FUNCTION_BLOCK FB_LogicSupply
VAR_IN_OUT
	bSwitchOn		: BOOL;
END_VAR

{attribute 'TcRpcEnable'}
METHOD SwitchOff
bSwitchOn := FALSE;
END_METHOD

{attribute 'TcRpcEnable'}
METHOD SwitchOn
bSwitchOn := TRUE;
END_METHOD

END_FUNCTION_BLOCK

(* stored: Version 1.1.0.1, ProductVersion 3.1.4024.11
   POU FB_LogicSupply: Id {ff82c6a0-8dc1-4585-a18c-a3c5cefd7a13}, SpecialFunc None
   Method SwitchOff: Id {9c28f1b0-2201-485b-9b73-f8448b8b551d}
   Method SwitchOn: Id {5e0e38e2-5b1a-46a2-b542-f19d9f565a0d} *)
